{attribute 'reflection'} 
FUNCTION_BLOCK FB_Event IMPLEMENTS I_Event
VAR_INPUT
	iLogger:					I_Logger;
END_VAR
VAR_OUTPUT
	fbArguments:				FB_Argument;
END_VAR
VAR
    {attribute 'hide'} 
    {attribute 'instance-path'} 
    {attribute 'noinit'} 
    sInstancePath:				STRING(255);
	fbSymbolInfo: 				PLC_ReadSymInfoByNameEx;
	fbVerbose:					FB_Message;
	fbInfo:						FB_Message;
	fbWarning:					FB_Message;
	fbError:					FB_Message;
	fbCritical:					FB_Message;
	stArchive:					ST_Events;

END_VAR

fbSymbolInfo();


// all events stay alive until mehtod is not called any more

IF fbVerbose.nTimestamp <> 0 THEN
	fbVerbose.nTimestamp:= 0;
ELSE
	fbVerbose.bActive:= FALSE;
END_IF

IF fbInfo.nTimestamp <> 0 THEN
	fbInfo.nTimestamp:= 0;
ELSE
	fbInfo.bActive:= FALSE;
END_IF

IF fbWarning.nTimestamp <> 0 THEN
	fbWarning.nTimestamp:= 0;
ELSE
	fbWarning.bActive:= FALSE;
END_IF

IF fbError.nTimestamp <> 0 THEN
	fbError.nTimestamp:= 0;
ELSE
	fbError.bActive:= FALSE;
END_IF

IF fbCritical.nTimestamp <> 0 THEN
	fbCritical.nTimestamp:= 0;
ELSE
	fbCritical.bActive:= FALSE;
END_IF

//FB_Init ist immer implizit verfügbar und wird primär für die Initialisierung verwendet.
//Der Rückgabewert wird nicht ausgewertet. Für gezielte Einflussnahme können Sie
//die Methoden explizit deklarieren und darin mit dem Standard-Initialisierungscode 
//zusätzlichen Code bereitstellen. Sie können den Rückgabewert auswerten.
METHOD FB_Init: BOOL
VAR_INPUT    
bInitRetains: BOOL; // TRUE: Die Retain-Variablen werden initialisiert (Reset warm / Reset kalt)    
bInCopyCode: BOOL:= True;  // TRUE: Die Instanz wird danach in den Kopiercode kopiert (Online-Change)
END_VAR
fbSymbolInfo.SYMNAME:= F_InstancePath(sInstancePath);
fbSymbolInfo.PORT:= TwinCAT_SystemInfoVarList._AppInfo.AdsPort;
fbSymbolInfo.START:= TRUE;
END_METHOD

METHOD PUBLIC M_Critical : BOOL
VAR_INPUT
	nID:				UDINT;
	sMessage:			STRING(255);
END_VAR
fbCritical.eLogLevel:= E_LogLevel.Critical;
fbCritical.nID:= nID;
fbCritical.nTimestamp:= F_GetSystemTime();
fbCritical.sMessage:= sMessage;
fbCritical.sArguments:= fbArguments.P_Value;
fbCritical.sDefault:= F_Print(sMessage, fbArguments.P_Value);
fbCritical.sSource:= fbSymbolInfo.SYMNAME;
fbCritical.sType:= fbSymbolInfo.SYMINFO.symDataType;

IF iLogger = 0 THEN
	F_Log(fbCritical);
ELSE
	iLogger.M_Log(fbCritical);
END_IF

fbArguments.M_Clear();
END_METHOD

METHOD PUBLIC M_Error : BOOL
VAR_INPUT
	nID:				UDINT;
	sMessage:			STRING(255);
END_VAR
fbError.eLogLevel:= E_LogLevel.Error;
fbError.nID:= nID;
fbCritical.nTimestamp:= F_GetSystemTime();
fbError.sMessage:= sMessage;
fbError.sArguments:= fbArguments.P_Value;
fbError.sDefault:= F_Print(sMessage, fbArguments.P_Value);
fbError.sSource:= fbSymbolInfo.SYMNAME;
fbError.sType:= fbSymbolInfo.SYMINFO.symDataType;

IF iLogger = 0 THEN
	F_Log(fbError);
ELSE
	iLogger.M_Log(fbError);
END_IF

fbArguments.M_Clear();
END_METHOD

METHOD PUBLIC M_Info : BOOL
VAR_INPUT
	nID:				UDINT;
	sMessage:			STRING(255);
END_VAR
fbInfo.eLogLevel:= E_LogLevel.Info;
fbInfo.nID:= nID;
fbInfo.nTimestamp:= F_GetSystemTime();
fbInfo.sMessage:= sMessage;
fbInfo.sArguments:= fbArguments.P_Value;
fbInfo.sDefault:= F_Print(sMessage, fbArguments.P_Value);
fbInfo.sSource:= fbSymbolInfo.SYMNAME;
fbInfo.sType:= fbSymbolInfo.SYMINFO.symDataType;

IF iLogger = 0 THEN
	F_Log(fbInfo);
ELSE
	iLogger.M_Log(fbInfo);
END_IF

fbArguments.M_Clear();
END_METHOD

METHOD PUBLIC M_Verbose : BOOL
VAR_INPUT
	sMessage:			STRING(255);
END_VAR
fbVerbose.eLogLevel:= E_LogLevel.Verbose;
fbVerbose.nID:= 0;
fbVerbose.nTimestamp:= F_GetSystemTime();
fbVerbose.sMessage:= sMessage;
fbVerbose.sArguments:= fbArguments.P_Value;
fbVerbose.sDefault:= F_Print(sMessage, fbArguments.P_Value);
fbVerbose.sSource:= fbSymbolInfo.SYMNAME;
fbVerbose.sType:= fbSymbolInfo.SYMINFO.symDataType;

IF iLogger = 0 THEN
	F_Log(fbVerbose);
ELSE
	iLogger.M_Log(fbVerbose);
END_IF

fbArguments.M_Clear();
END_METHOD

METHOD PUBLIC M_Warning : BOOL
VAR_INPUT
	nID:				UDINT;
	sMessage:			STRING(255);
END_VAR
fbWarning.eLogLevel:= E_LogLevel.Warning;
fbWarning.nID:= nID;
fbWarning.nTimestamp:= F_GetSystemTime();
fbWarning.sMessage:= sMessage;
fbWarning.sArguments:= fbArguments.P_Value;
fbWarning.sDefault:= F_Print(sMessage, fbArguments.P_Value);
fbWarning.sSource:= fbSymbolInfo.SYMNAME;
fbWarning.sType:= fbSymbolInfo.SYMINFO.symDataType;

IF iLogger = 0 THEN
	F_Log(fbWarning);
ELSE
	iLogger.M_Log(fbWarning);
END_IF

fbArguments.M_Clear();
END_METHOD

PROPERTY PUBLIC P_Argument : I_Argument
GET
P_Argument:= fbArguments;
END_GET
END_PROPERTY

PROPERTY PUBLIC P_Logger : I_Logger
GET
P_Logger:= iLogger;
END_GET
SET
iLogger:= P_Logger;
END_SET
END_PROPERTY

END_FUNCTION_BLOCK

(* stored: Version 1.1.0.1
   POU FB_Event: Id {fcfa56ff-d0f1-4149-9de7-6f44354915c6}, SpecialFunc None
   Method FB_Init: Id {256fe292-0b03-4593-83b5-0da540634dee}
   Method M_Critical: Id {7b4c91bf-8e3c-413c-a148-e271617106d9}
   Method M_Error: Id {11687e23-ea95-4e4f-aed4-4799ffa1ad84}
   Method M_Info: Id {7a920e55-da6d-473b-9aba-119c4de007e0}
   Method M_Verbose: Id {db95e385-16ed-493b-a6a5-28cc6625776b}
   Method M_Warning: Id {1aa0d3ef-0f74-4102-97d7-7d587822db85}
   Property P_Argument: Id {dd3bce54-33d7-4a6c-8d06-ad6a5d0ec566}
   Get Get: Id {9148b4be-b1fa-4fe4-a389-e96c939bba14}
   Property P_Logger: Id {98c079df-4944-4aae-a3d6-ca12ac41d1d4}
   Get Get: Id {7f49254e-94b6-4972-a1b5-02a92d10e780}
   Set Set: Id {4bbb606c-4053-49cc-ae04-84e1809ace25} *)
